FUNCTION_BLOCK FB_ESTOP_RESET
VAR_INPUT
END_VAR
VAR_OUTPUT
END_VAR
VAR
	
END_VAR

END_FUNCTION_BLOCK

(* stored: Version 1.1.0.1, ProductVersion 3.1.4024.12
   POU FB_ESTOP_RESET: Id {47ccba85-8c57-43fd-bb31-743461d2d675}, SpecialFunc None *)
